// TwinCAT 3 PLC project Untitled1
// ProgramVersion: 3.1.4023.0
// libraries:
//   Tc2_Standard, * (Beckhoff Automation GmbH)
//   Tc2_System, * (Beckhoff Automation GmbH)
//   Tc3_Module, * (Beckhoff Automation GmbH)
// project tree:
//   / GlobalTextList.TcGTLO, PlcTask.TcTTO, Visualization Manager.TcVMO (not stored)
//   GVLs/ button.TcDUT, sys_stat.TcDUT, enum_switch.TcDUT, joystick.TcPOU, vir_man_status.TcDUT, Visualization.TcVIS
//   POUs/ if_controller.TcIO, MAIN.TcPOU, ardu_map.TcPOU, POU.TcPOU, viritual_control_box.TcPOU, vir_man_switch.TcPOU
//   VISUs/ GVL.TcGVL, visual_box_GVL.TcGVL

CONFIGURATION Untitled1
    RESOURCE PLC ON TwinCAT3
        TASK PlcTask(INTERVAL := T#10ms, PRIORITY := 20);
        PROGRAM MAIN WITH PlcTask : MAIN;
    END_RESOURCE
END_CONFIGURATION

// ---- GVLs/button.TcDUT
{attribute 'qualified_only'}
{attribute 'strict'}
TYPE button :
(
	off := 0,
	on := 1
);
END_TYPE

// ---- GVLs/sys_stat.TcDUT
{attribute 'qualified_only'}
{attribute 'strict'}
TYPE sys_stat :
(
	notReady := 0,
	ready := 1,
	starting := 2,
	running := 3,
	stopping := 4,
	fault := 5
);
END_TYPE

// ---- GVLs/enum_switch.TcDUT
{attribute 'qualified_only'}
{attribute 'strict'}
TYPE enum_switch :
(
	off := 0,
	manual := 1,
	auto := 2
);
END_TYPE

// ---- GVLs/vir_man_status.TcDUT
{attribute 'qualified_only'}
{attribute 'strict'}
TYPE vir_man_status :
(
	virtual_box := 0,
	real_box := 1
);
END_TYPE

// ---- VISUs/GVL.TcGVL
{attribute 'qualified_only'}
VAR_GLOBAL
	startButton : button;
	stopButton : button;
	start_Button : BOOL;
	stop_Button : BOOL;
	mode_button : enum_switch := 0;
	rotSwitch : BOOL;
	vir_man_indi : vir_man_status;
END_VAR

// ---- VISUs/visual_box_GVL.TcGVL
{attribute 'qualified_only'}
VAR_GLOBAL
	start_button : BOOL;
	stop_button : BOOL;
	auto_button : BOOL;
	manual_button : BOOL;
	joy_x : LREAL;
	joy_y : LREAL;
	joy_button : BOOL;
END_VAR

// ---- POUs/if_controller.TcIO
INTERFACE if_controller

METHOD Mode
VAR_INPUT
	mode_stat : enum_switch;
END_VAR

METHOD Status
VAR_INPUT
	system_stat : sys_stat;
END_VAR

METHOD joystick
VAR_INPUT
	JOY_TopSwitch : BOOL;
	JOY_Y : REAL;
	Joy_X : REAL;
END_VAR

END_INTERFACE

// ---- POUs/MAIN.TcPOU
PROGRAM MAIN
VAR
	bEna : BOOL;
	bbbhei : BOOL;
	vir_mach : viritual_control_box;
	vir_stat : sys_stat;
	nu_val : LREAL := 1.1;
	su_val : LREAL;
	
	my_int : INT;
	my2_int : INT := 5;
	
	i_in_min : LREAL := 1000.0;
	i_in_max : LREAL := 2000.0;
	i_out_min : LREAL := 0;
	i_out_max : LREAL := 1.0;	
END_VAR

bEna := visual_box_GVL.auto_button;
vir_mach.status(current_sys_stat => vir_stat);
vir_stat;
ardu_map(in_val := visual_box_GVL.joy_x, in_min :=i_in_min, in_max := i_in_max, out_max := i_out_max, out_min := i_out_min, out_val => nu_val, mid_val => su_val);
nu_val;
su_val;
my_int := POU(int_in := my2_int);

END_PROGRAM

// ---- POUs/viritual_control_box.TcPOU
FUNCTION_BLOCK viritual_control_box //IMPLEMENTS if_controller
VAR_INPUT
END_VAR
VAR_OUTPUT
END_VAR
VAR
END_VAR

METHOD joystick : REAL
VAR_INPUT
END_VAR
END_METHOD

METHOD mode : enum_switch
VAR_INPUT
END_VAR
END_METHOD

METHOD status : sys_stat
VAR_INPUT
END_VAR
VAR_OUTPUT
	current_sys_stat : sys_stat;
END_VAR
VAR
	have_start_been_high : BOOL := FALSE;
	have_stop_been_high : BOOL := FALSE;
END_VAR
IF GVL.start_Button = TRUE THEN
	current_sys_stat := sys_stat.ready;
ELSIF GVL.start_Button = FALSE THEN
	current_sys_stat := sys_stat.fault;
ELSE
	current_sys_stat := sys_stat.notReady;
END_IF
END_METHOD

END_FUNCTION_BLOCK

// ---- GVLs/joystick.TcPOU
FUNCTION_BLOCK joystick
VAR_INPUT
END_VAR
VAR_OUTPUT
END_VAR
VAR
END_VAR

END_FUNCTION_BLOCK

// ---- POUs/ardu_map.TcPOU
FUNCTION ardu_map : LREAL
VAR_INPUT
	in_val : LREAL;
	in_min : LREAL;
	in_max : LREAL;
	out_min : LREAL;
	out_max : LREAL;
END_VAR
VAR
END_VAR
VAR_OUTPUT
	out_val : LREAL;
	mid_val : LREAL;
END_VAR

in_max := mid_val;
out_val := (in_val - in_min) * (out_max - out_min) / (in_max - in_min) + out_min;

//(x - in_min) * (out_max - out_min) / (in_max - in_min) + out_min;

END_FUNCTION

// ---- POUs/POU.TcPOU
FUNCTION POU : INT
VAR_INPUT
	int_in : INT;
END_VAR
VAR
END_VAR

POU := int_in;

END_FUNCTION

// ---- POUs/vir_man_switch.TcPOU
FUNCTION_BLOCK vir_man_switch
VAR_INPUT
	vir_real_trig : BOOL;
END_VAR
VAR_OUTPUT
END_VAR
VAR
END_VAR

IF vir_real_trig := TRUE THEN
	GVL.vir_man_indi := vir_man_status.real_box;
ELSE
	GVL.vir_man_indi := vir_man_status.virtual_box;
END_IF

END_FUNCTION_BLOCK

// ---- GlobalTextList.TcGTLO
TEXTLIST GlobalTextList
  352 = 'auto'
  257 = 'Control box'
  67 = 'manuel'
  483 = 'start'
  632 = 'stop'
END_TEXTLIST

// ---- GVLs/Visualization.TcVIS
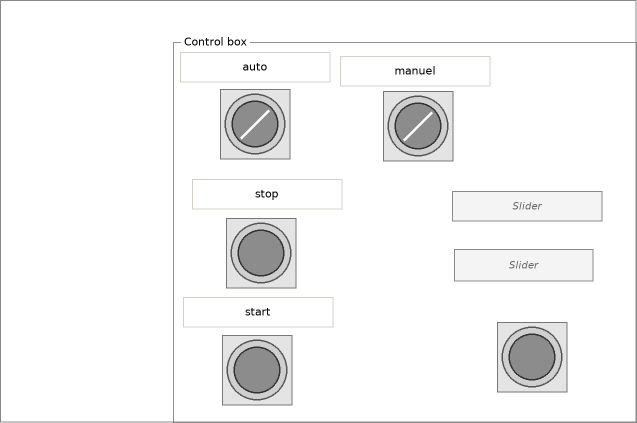
VISUALIZATION Visualization  // 637x423
    GroupBox (173,34 464x389), "Control box"
        PushSwitch (53,184 70x70), variable: visual_box_GVL.stop_button, behaviour: TOGGLE, style: Switch-PushSwitch-Gray
        PushSwitch (49,301 70x70), variable: visual_box_GVL.start_button, behaviour: TOGGLE, style: Switch-PushSwitch-Gray
        RotarySwitch (210,57 70x70), variable: visual_box_GVL.manual_button, behaviour: TOGGLE, style: Switch-RotarySwitch-Gray
        RotarySwitch (47,55 70x70), variable: visual_box_GVL.auto_button, behaviour: TOGGLE, style: Switch-RotarySwitch-Gray
        Slider (279,157 150x30), variable: visual_box_GVL.joy_x, scale 1000..2000
        Slider (281,215 139x32), variable: visual_box_GVL.joy_y, scale 1100..1900
        PushSwitch (324,288 70x70), variable: visual_box_GVL.joy_button, behaviour: TOGGLE, style: Switch-PushSwitch-Gray
        Textfield (10,263 150x30), "start"
        Textfield (167,22 150x30), "manuel"
        Textfield (19,145 150x30), "stop"
        Textfield (7,18 150x30), "auto"
END_VISUALIZATION
